FUNCTION_BLOCK RingTokenCTL (* Basic Function Block Type *)
  (* Standard: 61499-2 *)
  (* Version 0.2, 2003-12-04, JHC, Rockwell Automation, Renamed for better indexing. *)
  (* Version 0.1, 2002-11-05, JHC, Rockwell Automation, Corrected missing ST element in Algorithm REQ. *)
  (* Version 0.0, 2000-05-30, JHC, Rockwell Automation *)
  (* Compiler header: package fb.rt.cs725; *)
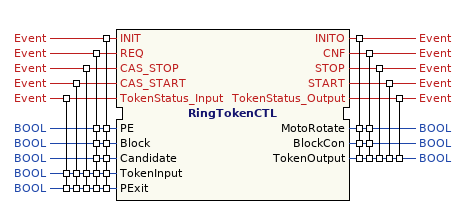
  EVENT_INPUT
    INIT WITH PE, Block, Candidate, TokenInput, PExit; (* Initialization Request *)
    REQ WITH PE, Block, Candidate, TokenInput, PExit; (* Normal Execution Request *)
    CAS_STOP WITH TokenInput, PExit;
    CAS_START WITH TokenInput, PExit;
    TokenStatus_Input WITH TokenInput, PExit;
  END_EVENT
  EVENT_OUTPUT
    INITO WITH MotoRotate, BlockCon, TokenOutput; (* Initialization Confirm *)
    CNF WITH MotoRotate, BlockCon, TokenOutput; (* Execution Confirmation *)
    STOP WITH TokenOutput;
    START WITH TokenOutput;
    TokenStatus_Output WITH TokenOutput;
  END_EVENT
  VAR_INPUT
    PE : BOOL; (* Input event qualifier *)
    Block : BOOL;
    Candidate : BOOL;
    TokenInput : BOOL;
    PExit : BOOL;
  END_VAR
  VAR_OUTPUT
    MotoRotate : BOOL; (* Output event qualifier *)
    BlockCon : BOOL;
    TokenOutput : BOOL;
  END_VAR
  VAR
    lastPE : BOOL := 1;
    lastBlock : BOOL := 0;
  END_VAR
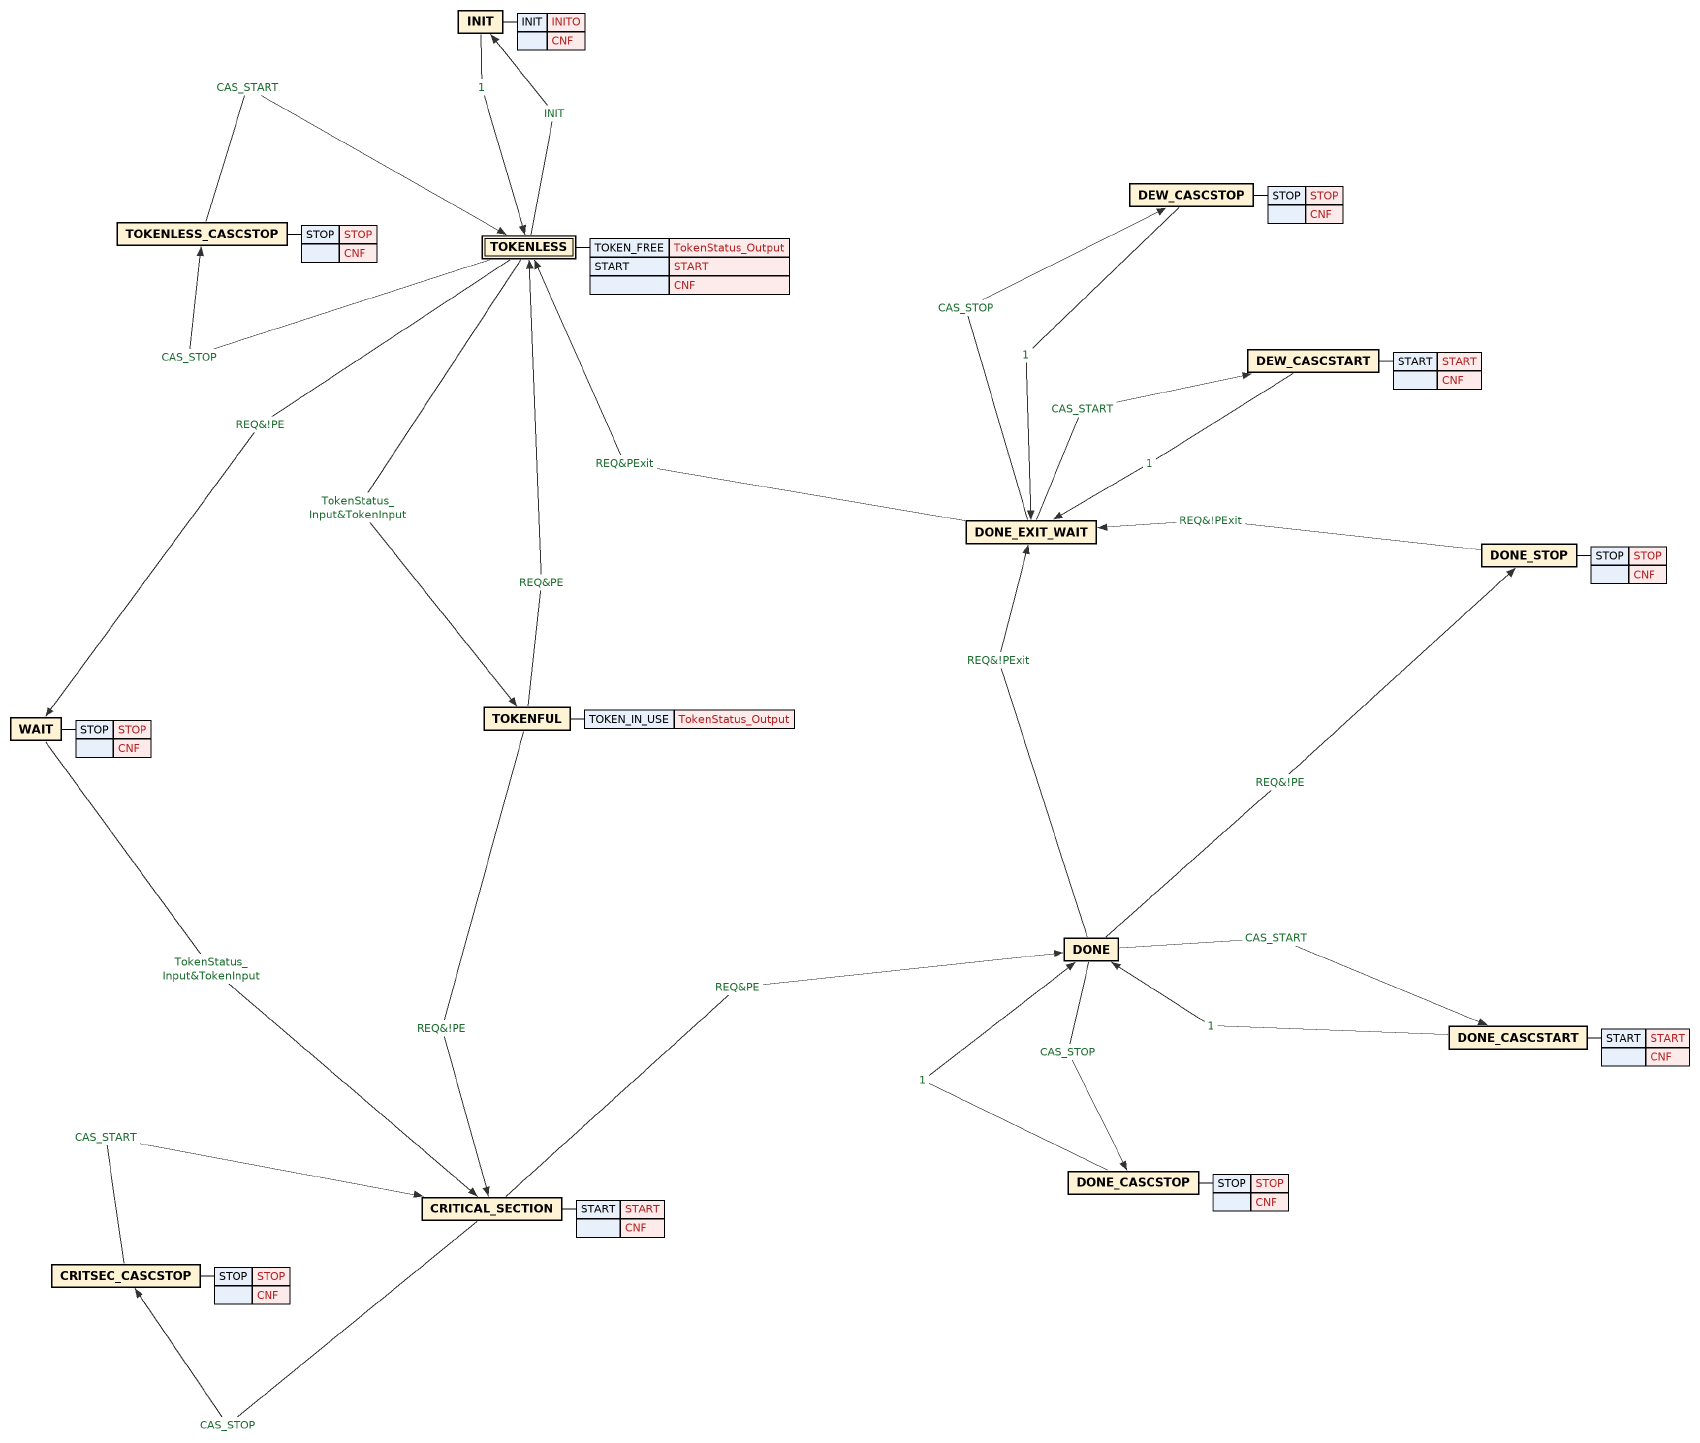
  EC_STATES
    TOKENLESS : TOKEN_FREE -> TokenStatus_Output, START -> START, -> CNF; (* Doesn't have the token *)
    INIT : INIT -> INITO, -> CNF; (* Initialization *)
    WAIT : STOP -> STOP, -> CNF; (* waiting for token *)
    TOKENFUL : TOKEN_IN_USE -> TokenStatus_Output;
    CRITICAL_SECTION : START -> START, -> CNF; (* Entering the critical section *)
    DONE; (* Leaving critical section *)
    DONE_STOP : STOP -> STOP, -> CNF; (* If another one comes behind then stop the conveyor *)
    DONE_EXIT_WAIT;
    TOKENLESS_CASCSTOP : STOP -> STOP, -> CNF;
    CRITSEC_CASCSTOP : STOP -> STOP, -> CNF;
    DONE_CASCSTOP : STOP -> STOP, -> CNF;
    DONE_CASCSTART : START -> START, -> CNF;
    DEW_CASCSTOP : STOP -> STOP, -> CNF;
    DEW_CASCSTART : START -> START, -> CNF;
  END_STATES
  EC_TRANSITIONS
    INIT TO TOKENLESS := 1;
    TOKENLESS TO WAIT := REQ&!PE; (* tick and photoeye sensor *)
    WAIT TO CRITICAL_SECTION := TokenStatus_Input&TokenInput; (* token status changed nd token availabale *)
    TOKENFUL TO CRITICAL_SECTION := REQ&!PE; (* needs token so go into critical section *)
    TOKENLESS TO TOKENFUL := TokenStatus_Input&TokenInput; (* receives the token *)
    TOKENFUL TO TOKENLESS := REQ&PE; (* Token not needed *)
    CRITICAL_SECTION TO DONE := REQ&PE; (* No longer being sensed by photo eye *)
    TOKENLESS TO INIT := INIT;
    DONE TO DONE_STOP := REQ&!PE;
    DONE TO DONE_EXIT_WAIT := REQ&!PExit;
    DONE_STOP TO DONE_EXIT_WAIT := REQ&!PExit;
    DONE_EXIT_WAIT TO TOKENLESS := REQ&PExit;
    TOKENLESS TO TOKENLESS_CASCSTOP := CAS_STOP;
    TOKENLESS_CASCSTOP TO TOKENLESS := CAS_START;
    CRITICAL_SECTION TO CRITSEC_CASCSTOP := CAS_STOP;
    CRITSEC_CASCSTOP TO CRITICAL_SECTION := CAS_START;
    DONE TO DONE_CASCSTOP := CAS_STOP;
    DONE_CASCSTOP TO DONE := 1;
    DONE TO DONE_CASCSTART := CAS_START;
    DONE_CASCSTART TO DONE := 1;
    DONE_EXIT_WAIT TO DEW_CASCSTOP := CAS_STOP;
    DEW_CASCSTOP TO DONE_EXIT_WAIT := 1;
    DONE_EXIT_WAIT TO DEW_CASCSTART := CAS_START;
    DEW_CASCSTART TO DONE_EXIT_WAIT := 1;
  END_TRANSITIONS
  ALGORITHM INIT IN ST: (* Initialization algorithm *)
MotoRotate := TRUE;
Block := FALSE;

System.out.println(this + " " + MotoRotate);
System.out.println(MotoRotate);
  END_ALGORITHM
  ALGORITHM REQ IN ST: (* Normally executed algorithm *)
System.out.println(this +  " -> Candidate" + Candidate);
IF Candidate THEN
IF lastPE !:= PE THEN
IF NOT PE THEN
BlockCon:= TRUE;
System.out.println("BlockCon = true");
ELSE
BlockCon:=FALSE;
System.out.println("BlockCon = false");
END_IF
lastPE := PE;
END_IF
IF lastBlock !:= Block THEN
IF Block THEN
STOP.serviceEvent(this);
MotoRotate := FALSE;
System.out.println("Cas Stop");
ELSE
START.serviceEvent(this);
MotoRotate := TRUE;
System.out.println("Cas Start");
END_IF
lastBlock := Block;
END_IF
END_IF
  END_ALGORITHM
  ALGORITHM START IN ST:
MotoRotate:=TRUE;
System.out.println(this + " Start " + MotoRotate);

System.out.println("Start " + MotoRotate);
  END_ALGORITHM
  ALGORITHM STOP IN ST:
MotoRotate := FALSE;
System.out.println(this + " Stop " + MotoRotate);

System.out.println("Stop " + MotoRotate);
  END_ALGORITHM
  ALGORITHM TOKEN_IN_USE IN ST:
TokenOutput := FALSE;
  END_ALGORITHM
  ALGORITHM TOKEN_FREE IN ST:
TokenOutput := TRUE;
  END_ALGORITHM
END_FUNCTION_BLOCK
